FUNCTION_BLOCK EP3751_Accelerometer EXTENDS CyclicComponent
VAR
    

END_VAR

END_FUNCTION_BLOCK

(* stored: Version 1.1.0.1
   POU EP3751_Accelerometer: Id {f8ec9d09-616a-4dab-9965-542afba73c73}, SpecialFunc None *)
